# EPICS autosave request: GALIL/iocBoot/iocGALIL-IOC-04/GALIL_04_settings.req
file "GALIL_controller_settings.req" P=$(P),CCP=$(CCP)
